FUNCTION_BLOCK Test_DateAsString EXTENDS TUnitTestBase
VAR
END_VAR

METHOD  Execute
VAR_INST
    TimeStruct : TIMESTRUCT := (wDay := 23, wMonth := 12, wYear := 1945);
END_VAR
AssertEquals_STRING(
    Expected := '23/12/1945',
    Actual   := F_DateAsString(TimeStruct),
    VariableName  := 'F_DateAsString(TimeStruct)');


Test_Finished();
END_METHOD

END_FUNCTION_BLOCK

(* stored: Version 1.1.0.1, ProductVersion 3.1.4024.3
   POU Test_DateAsString: Id {dbb0c8d6-f694-0d2d-11c0-291b7b634d6f}, SpecialFunc None
   Method Execute: Id {515db551-4021-0c2c-26e7-a8eed9752a07} *)
